PROGRAM PersistentData
VAR
	
	FB_GetUPSStatus_0: FB_GetUPSStatus;
	FB_WritePersistent: FB_WritePersistentData;
	MODE :E_PersistentMode; 
	Status:ST_UPSStatus;
END_VAR
VAR // added by the converter: edge detectors and wires of the graphical bodies
    _w1 : BOOL;
    _w2 : ANY;
END_VAR

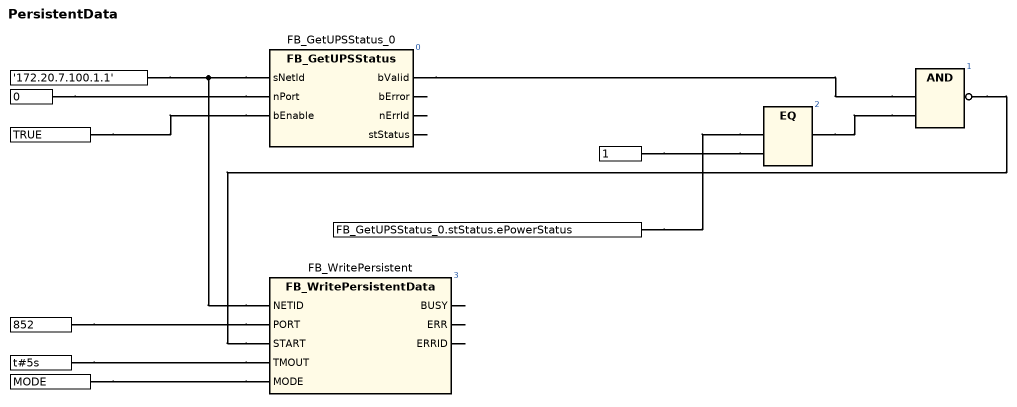
FB_GetUPSStatus_0(sNetId := '172.20.7.100.1.1', nPort := 0, bEnable := TRUE); // FB_GetUPSStatus
_w2 := FB_GetUPSStatus_0.bValid AND _w1;
_w1 := FB_GetUPSStatus_0.stStatus.ePowerStatus = 1;
FB_WritePersistent(NETID := '172.20.7.100.1.1', PORT := 852, START := NOT _w2, TMOUT := t#5s, MODE := MODE); // FB_WritePersistentData

END_PROGRAM

(* stored: Version 1.1.0.1, ProductVersion 3.1.4020.12
   POU PersistentData: Id {e68f672f-ba27-41dd-a512-d8613b2736dc}, SpecialFunc None *)
